{attribute 'no_explicit_call':= 'do not call this POU directly'}
FUNCTION_BLOCK T_ValueMonitor
VAR
    _CurrentValue  : INT := -1;
    _PreviousValue : INT;
    _Changed       : BOOL;
END_VAR

PROPERTY Changed : BOOL
GET
Changed := _Changed;
END_GET
END_PROPERTY

PROPERTY CurrentValue : INT
GET
CurrentValue := _CurrentValue;
END_GET
END_PROPERTY

PROPERTY PreviousValue : INT
GET
PreviousValue := _PreviousValue;
END_GET
END_PROPERTY

METHOD Reset
VAR_INPUT
END_VAR
_CurrentValue  := 0;
_PreviousValue := 0;
END_METHOD

METHOD Test : BOOL
VAR_INPUT
    Value : INT;
END_VAR
_Changed       := Value <> _CurrentValue;
_PreviousValue := _CurrentValue;
_CurrentValue  := Value;

Test := _Changed;
END_METHOD

END_FUNCTION_BLOCK

(* stored: Version 1.1.0.1, ProductVersion 3.1.4024.12
   POU T_ValueMonitor: Id {4b037847-6583-01a2-1bbd-221df4c80ab7}, SpecialFunc None
   Property Changed: Id {1b3df0f3-95f2-07b0-013f-91fdb932be9f}
   Get Get: Id {cbd42d68-ba9d-0857-2253-cff857dc47d0}
   Property CurrentValue: Id {65539bed-a55c-0c12-1fb0-72168bc8bb67}
   Get Get: Id {3aa6fe1c-a4aa-04b6-33da-dfe6cc8defbf}
   Property PreviousValue: Id {d60a3b17-98a8-0704-0cd8-a6f1ee361aea}
   Get Get: Id {a6e558fb-1618-0abb-0e12-7d0a966298f1}
   Method Reset: Id {867e6174-75fd-07d3-3cff-4113b2c8edfa}
   Method Test: Id {101a9467-dca8-0219-3b89-c70c9469009d} *)
